// TIA Portal V16 export
// export: Created 2022-02-04T14:40:18.912128Z, ExportSetting WithDefaults, DisplayName Totally Integrated Automation Portal, DisplayVersion V16 Update 1, DisplayName TIA Portal Version Control Interface, DisplayVersion V16, DisplayName TIA Portal Openness, DisplayVersion V16, DisplayName SINAMICS Startdrive Advanced, DisplayVersion V16 Update 5, DisplayName SINAMICS Startdrive G130, G150, S120, S150, SINAMICS MV, S210, DisplayVersion V16 Update 5, DisplayName SINAMICS Startdrive G110M, G120, G120C, G120D, G120P, G115D, DisplayVersion V16 Update 5, DisplayName STEP 7 Professional, DisplayVersion V16, DisplayName STEP 7 Safety, DisplayVersion V16, DisplayName WinCC Advanced, DisplayVersion V16, DisplayName SIMATIC Visualization Architect, DisplayVersion V16
DATA_BLOCK "IM_PFM"   // DB14
VERSION : 0.1
// stored: AutoNumber true, InstanceOfName FB_IM_PFM, InstanceOfType FB
"FB_IM_PFM"
   // VAR RETAIN
   //    M_233_Fork_PFM : "FB_IM2x4";
   //    M_232_Elevator_PFM { S7_SetPoint := 'True'} : "FB_IM2x2S";
   //    M_317_Gasket_Carousel { S7_SetPoint := 'True'} : "FB_IM2x1";
   //    Elevator_brake_timer { S7_SetPoint := 'True'} : TON;
   // END_VAR
BEGIN
   M_233_Fork_PFM.SpeedOn := 15.0;
   M_233_Fork_PFM.SpeedOnLow := 10.0;
   M_233_Fork_PFM.SpeedOff := 15.0;
   M_233_Fork_PFM.SpeedOffLow := 10.0;
END_DATA_BLOCK
